METHOD Start : BOOL
VAR_INPUT
END_VAR
bDone := FALSE;
step := 1;
END_METHOD

END_PROGRAM

// ---- POUs/功能塊/Stober驅動/ReadStoberError.TcPOU
PROGRAM ReadStoberError
VAR
	step: INT;
	
	raw_Data	: DWORD;
	
	fb_CoERead : FB_EcCoESdoRead;
	
	readindex : INT;
	
	i_Event :ARRAY [0..17] OF UDINT;
	i_CASE :ARRAY [0..17] OF UDINT;
	
	
	EtherCatAddr	: ARRAY [0..8] OF T_AmsNetId := [9('0.0.0.0.3.1')];
	DriverAddr		: ARRAY [0..8] OF UINT := [1010,1011,1012,1013,1014,1015,1017,1018,1019];
	MoterName		: ARRAY [0..17] OF WSTRING := ["Fx1", "Fx2", "Ax", "Ay", "Az1", "Az2", "Bx", "Bz", "By1", "By2", "Cz1", "Cz2", "Cx", "Cy", "Dy", "Dx", "Dz", "NA"];
	i: INT;
	
	showNumber 		: INT;
END_VAR

CASE step OF
	1:
		fb_CoERead.bExecute		:= FALSE;
		readindex := 0;
		step := step + 1;
		
	2:
		step := 10;
		
	10:
		fb_CoERead.sNetId		:= EtherCatAddr[readindex];
		fb_CoERead.nSlaveAddr	:= DriverAddr[readindex];
		fb_CoERead.nIndex		:= 16#2852;
		fb_CoERead.pDstBuf		:= ADR(raw_Data);
		fb_CoERead.cbBufLen		:= 4;
		fb_CoERead.bExecute		:= TRUE;
		step := step + 1;
		
	11:
		IF NOT fb_CoERead.bBusy THEN
			fb_CoERead.bExecute		:= FALSE;
			step := step + 1;
		END_IF
		
	12:
		IF NOT fb_CoERead.bError THEN
			i_Event[readindex * 2] := DWORD_TO_UDINT(raw_Data);
			step := step + 1;
		ELSE
			step := 0;
		END_IF
	
	13:
		raw_Data := 0;
		step := 20;
		
	20:
		fb_CoERead.nIndex		:= 16#282B;
		fb_CoERead.pDstBuf		:= ADR(raw_Data);
		fb_CoERead.cbBufLen		:= 4;
		fb_CoERead.bExecute		:= TRUE;
		step := step + 1;
		
	21:
		IF NOT fb_CoERead.bBusy THEN
			fb_CoERead.bExecute		:= FALSE;
			step := step + 1;
		END_IF
		
	22:
		IF NOT fb_CoERead.bError THEN
			i_CASE[readindex * 2] := DWORD_TO_UDINT(raw_Data);
			step := step + 1;
		ELSE
			step := 0;
		END_IF
	
	23:
		raw_Data := 0;
		step := 30;
		
	30:
		fb_CoERead.nIndex		:= 16#A852;
		fb_CoERead.pDstBuf		:= ADR(raw_Data);
		fb_CoERead.cbBufLen		:= 4;
		fb_CoERead.bExecute		:= TRUE;
		step := step + 1;
		
	31:
		IF NOT fb_CoERead.bBusy THEN
			fb_CoERead.bExecute		:= FALSE;
			step := step + 1;
		END_IF
		
	32:
		IF NOT fb_CoERead.bError THEN
			i_Event[readindex * 2 + 1] := DWORD_TO_UDINT(raw_Data);
			step := step + 1;
		ELSE
			step := 0;
		END_IF
	
	33:
		raw_Data := 0;
		step := 40;
		
	40:
		fb_CoERead.nIndex		:= 16#A82B;
		fb_CoERead.pDstBuf		:= ADR(raw_Data);
		fb_CoERead.cbBufLen		:= 4;
		fb_CoERead.bExecute		:= TRUE;
		step := step + 1;
		
	41:
		IF NOT fb_CoERead.bBusy THEN
			fb_CoERead.bExecute		:= FALSE;
			step := step + 1;
		END_IF
		
	42:
		IF NOT fb_CoERead.bError THEN
			i_CASE[readindex * 2 + 1] := DWORD_TO_UDINT(raw_Data);
			step := step + 1;
		ELSE
			step := 0;
		END_IF
	
	43:
		raw_Data := 0;
		step := 50;
		
	50:
		IF readindex < 5 THEN
		 	readindex := readindex + 1;
			step := 10;
		ELSE
			readindex := 0;
			step := step + 1;
		END_IF
		
	51:
		step := 60;
		
	60:
		IF showNumber > 0 AND showNumber <= 17 THEN
			i := showNumber - 1;
			step := 61;
		ELSE
			i := 0;
			step := 62;
		END_IF
		
	61:
		pMsg.Push_Info(ErrorCodeConver.StoberErrorCode(MoterName[i], i_Event[i], i_case[i]));
		pMsg.Push_Info(
			WCONCAT(
				STR1:= MoterName[i],
				STR2:= StoberErrorStr(i_Event[i], i_case[i])
		));
		step := 65;
		
	62:
		IF i < 12 AND i <> 8 AND i_Event[i] <> 30 THEN
			pMsg.Push_Info(ErrorCodeConver.StoberErrorCode(MoterName[i], i_Event[i], i_case[i]));
			pMsg.Push_Info(
				WCONCAT(
					STR1:= MoterName[i],
					STR2:= StoberErrorStr(i_Event[i], i_case[i])
			));
		END_IF
		step := step + 1;
		
	63:
		i := i + 1;
		IF i < 12 THEN
			step := step - 1;
		ELSE
			step := 65;
		END_IF
		
	65:
		i := 0;
		step := 90;
		
	90:
		step := 0;
END_CASE

fb_CoERead();

METHOD Read : BOOL
VAR_INPUT
	// 選擇軸
	Axis : AXIS_REF;
END_VAR

step := 1;
END_METHOD

END_PROGRAM

// ---- POUs/功能塊/Stober驅動/StoberErrorStr.TcPOU
FUNCTION StoberErrorStr : WSTRING
VAR_INPUT
	in_Event	: UDINT;
	in_Case		: UDINT;
END_VAR
VAR
END_VAR

CASE in_Event OF
	31:	
		StoberErrorStr := "Short/ground";
		
	32:	
		StoberErrorStr := "Short/ground internal";
		
	33:	
		CASE in_Case OF
			1:
				StoberErrorStr := "Overcurrent(Normal)";
			2:
				StoberErrorStr := "Overcurrent(Fast)";
		END_CASE
		
	34:
		CASE in_Case OF
			1,23,24,25:
				StoberErrorStr := "Hardware fault(FPGA)";
			2:
				StoberErrorStr := "Hardware fault(NOV control unit)";
			3:
				StoberErrorStr := "Hardware fault(NOV-Power Unit)";
			4,5:
				StoberErrorStr := "Hardware fault(Inactive)";
			6:
				StoberErrorStr := "Hardware fault(NOV safety module)";
			7:
				StoberErrorStr := "Hardware fault(Current measurement)";
			8,9,10,11,30:
				StoberErrorStr := "Hardware fault(power supply)";
			12:
				StoberErrorStr := "Hardware fault(Timer control board)";
			13:
				StoberErrorStr := "Hardware fault(Communication module adress-/databus)";
			14:
				StoberErrorStr := "Hardware fault(Communication module signal lines)";
			15:
				StoberErrorStr := "Hardware fault(Communication module clock error)";
			16:
				StoberErrorStr := "Hardware fault(Communication module voltage missing)";
			17:
				StoberErrorStr := "Hardware fault(Communication module databus)";
			18:
				StoberErrorStr := "Hardware fault(Terminal module adress-/databus)";
			19:
				StoberErrorStr := "Hardware fault(Terminal module signal lines)";
			20:
				StoberErrorStr := "Hardware fault(Terminal module clock error)";
			21:
				StoberErrorStr := "Hardware fault(Terminal module voltage is missing)";
			22:
				StoberErrorStr := "Hardware fault(Terminal module databus)";
			26,27,28:
				StoberErrorStr := "Hardware fault(CPU)";
			29:
				StoberErrorStr := "Hardware fault(Communication)";
			31:
				StoberErrorStr := "Hardware fault(Operating unit)";
		END_CASE
		
	35:	
		CASE in_Case OF
			1:
				StoberErrorStr := "Watchdog(Core 0)";
			2:
				StoberErrorStr := "Watchdog(Core 1)";
		END_CASE
		
	36:	
		StoberErrorStr := "High voltage";
		
	37:	
		CASE in_Case OF
			1:
				StoberErrorStr := "Motor encoder(Parameter <-> encoder)";
			2:
				StoberErrorStr := "Motor encoder(Maximum speed)";
			3,5:
				StoberErrorStr := "Motor encoder(AX6)";
			4:
				StoberErrorStr := "Motor encoder(Required AX6)";
			6:
				StoberErrorStr := "Motor encoder(X4 EnDat encoder found)";
			7:
				StoberErrorStr := "Motor encoder(X4 A track/Incremental)";
			8:
				StoberErrorStr := "Motor encoder(X4 no encoder found)";
			10:
				StoberErrorStr := "Motor encoder(X4 A track/Clk)";
			11:
				StoberErrorStr := "Motor encoder(X4 B track/Dat)";
			12:
				StoberErrorStr := "Motor encoder(X4 N track)";
			13:
				StoberErrorStr := "Motor encoder(X4-EnDat alarm)";
			14:
				StoberErrorStr := "Motor encoder(X4 EnDat CRC)";
			15:
				StoberErrorStr := "Motor encoder(X4 double transmission)";
			16:
				StoberErrorStr := "Motor encoder(X4 busy)";
			17:
				StoberErrorStr := "Motor encoder(EBI encoder low battery)";
			18:
				StoberErrorStr := "Motor encoder(EBI encoder battery empty)";
			19:
				StoberErrorStr := "Motor encoder(Alarm bit)";
			20:
				StoberErrorStr := "Motor encoder(Resolver carrier)";
			21:
				StoberErrorStr := "Motor encoder(Low voltage)";
			22:
				StoberErrorStr := "Motor encoder(Resolver sin/cos overvoltage)";
			23,24:
				StoberErrorStr := "Motor encoder(Resolver failure)";
			30:
				StoberErrorStr := "Motor encoder(X120 wire break)";
			35:
				StoberErrorStr := "Motor encoder(X120 double transmission)";
			36:
				StoberErrorStr := "Motor encoder(X120 busy)";
			38:
				StoberErrorStr := "Motor encoder(X120 timeout)";
			43:
				StoberErrorStr := "Motor encoder(X140 EnDat alarm)";
			44:
				StoberErrorStr := "Motor encoder(X140 EnDat CRC)";
			48:
				StoberErrorStr := "Motor encoder(X4 zero pulse missing)";
			49:
				StoberErrorStr := "Motor encoder(X4 zero pulse distance too small)";
			60:
				StoberErrorStr := "Motor encoder(Hiperface synchronisation)";
			61:
				StoberErrorStr := "Motor encoder(Hiperface timeout)";
			62:
				StoberErrorStr := "Motor encoder(Hiperface signal quality)";
			63:
				StoberErrorStr := "Motor encoder(Hiperface link)";
			64:
				StoberErrorStr := "Motor encoder(EnDat3 Timeout)";
			65:
				StoberErrorStr := "Motor encoder(EnDat3 invalid Request)";
			66:
				StoberErrorStr := "Motor encoder(EnDat3 Position Check)";
		END_CASE
		
	38:	
		StoberErrorStr := "Temperature drive controller sensor";
	39:	
		StoberErrorStr := "Temperature drive controller sensor";
		
	40:
		CASE in_Case OF
			1:
				StoberErrorStr := "Invalid data(Fault)";
			2,7:
				StoberErrorStr := "Invalid data(Block missing)";
			3:
				StoberErrorStr := "Invalid data(Data security)";
			4:
				StoberErrorStr := "Invalid data(Checksum)";
			5:
				StoberErrorStr := "Invalid data(Read only)";
			6:
				StoberErrorStr := "Invalid data(Read error)";
			8:
				StoberErrorStr := "Invalid data(Wrong/illegal serial number)";
			9:
				StoberErrorStr := "Invalid data(A00 interrupted - data loss)";
			32:
				StoberErrorStr := "Invalid data(Electronic nameplate)";
			33:
				StoberErrorStr := "Invalid data(Electronic nameplate limit)";
			48:
				StoberErrorStr := "Invalid data(Reverse documentation)";
		END_CASE
		
	41:
		StoberErrorStr := "Temp.MotorTMP";
	24:
		StoberErrorStr := "TempBrakeRes";
	43:
		StoberErrorStr := "AI1 wire break";
	44:
		StoberErrorStr := "External fault 1";
	45:
		StoberErrorStr := "Overtemp.motor i2t";
	46:
		CASE in_Case OF
			1:
				StoberErrorStr := "Low voltage(DC link voltage below limit)";
			2:
				StoberErrorStr := "Low voltage(Failure of one/ all phases (mains))";
			3:
				StoberErrorStr := "Low voltage(Drop in network voltage when power section active)";
		END_CASE
	
	47:
		StoberErrorStr := "Torque/force-max. limit";
	48:
		StoberErrorStr := "Brake release monitoring";
	49:
		CASE in_Case OF
			1:
				StoberErrorStr := "Brake(Brake supply voltage too low)";
			2:
				StoberErrorStr := "Brake(Brake 1: no feedback)";
			3:
				StoberErrorStr := "Brake(Brake 1: short circuit)";
			4:
				StoberErrorStr := "Brake(Brake 1: open load)";
			5:
				StoberErrorStr := "Brake(Brake 2: no feedback)";
			6:
				StoberErrorStr := "Brake(Brake 2: short circuit)";
			7:
				StoberErrorStr := "Brake(Brake 2: open load)";
			8:
				StoberErrorStr := "Brake(F92 switchover not permitted for opened brake)";
			9:
				StoberErrorStr := "Brake(Brake 1 slips)";
			10:
				StoberErrorStr := "Brake(Brake monitoring with engaged brake)";
			11:
				StoberErrorStr := "Brake(Brake monitoring with released brake)";
			12:
				StoberErrorStr := "Brake(Brake monitoring during engaging time)";
			13:
				StoberErrorStr := "Brake(Brake monitoring during release time)";
		END_CASE
	50:
		CASE in_Case OF
			1:
				StoberErrorStr := "Safety module(Inconsistent request (single channel))";
			2:
				StoberErrorStr := "Safety module(Wrong safety module)";
			3:
				StoberErrorStr := "Safety module(Internal error)";
			4:
				StoberErrorStr := "Safety module(PowerUp sequence error)";
			5:
				StoberErrorStr := "Safety module(Wrong interface version)";
			6:
				StoberErrorStr := "Safety module(Fatal error)";
			7:
				StoberErrorStr := "Safety module(Different CRCs in safety config of SafetyModule and DS6)";
			8:
				StoberErrorStr := "Safety module(Safety module startup error)";
			9:
				StoberErrorStr := "Safety module(Safety module failure)";
			10:
				StoberErrorStr := "Safety module(Safety config. missing in ParaModul)";
			11:
				StoberErrorStr := "Safety module(Safety config. from ParaModul activated)";
			12:
				StoberErrorStr := "Safety module(Safety config. missing in Paramodul&safety module)";
			13:
				StoberErrorStr := "Safety module(Safety module activation error)";
			14:
				StoberErrorStr := "Safety module(Command drive to safety module timeout)";
			15:
				StoberErrorStr := "Safety module(Safety module error)";
			16:
				StoberErrorStr := "Safety module(Remove enable!)";
			17:
				StoberErrorStr := "Safety module(Error class LIMIT)";
			18:
				StoberErrorStr := "Safety module(Error class OTHER)";
			19:
				StoberErrorStr := "Safety module(Safety module invalid FSoE address)";
			20:
				StoberErrorStr := "Safety module(Safety control word Error)";
		END_CASE
	51:
		CASE in_Case OF
			1:
				StoberErrorStr := "Virtual master software limit switch(SW-limit switch positive)";
			2:
				StoberErrorStr := "Virtual master software limit switch(SW-limit switch negative)";
			3:
				StoberErrorStr := "Virtual master software limit switch(+/- 31 bit computing limit reached)";
		END_CASE
	52:
		CASE in_Case OF
			1:
				StoberErrorStr := "Communication(CAN Life Guarding Event)";
			2:
				StoberErrorStr := "Communication(CAN Sync Error)";
			3:
				StoberErrorStr := "Communication(CAN Bus Off)";
			4:
				StoberErrorStr := "Communication(PZD-Timeout)";
			5:
				StoberErrorStr := "Communication(Wrong or missing X3 firmware)";
			6:
				StoberErrorStr := "Communication(EtherCAT PDO-Timeout)";
			7:
				StoberErrorStr := "Communication(Reserved)";
			8:
				StoberErrorStr := "Communication(IGB µC failure)";
			9:
				StoberErrorStr := "Communication(IGB serie lost frames)";
			10:
				StoberErrorStr := "Communication(IGB partner serie lost frames)";
			11:
				StoberErrorStr := "Communication(IGB synchronization error)";
			12:
				StoberErrorStr := "Communication(IGB configuration timing)";
			13:
				StoberErrorStr := "Communication(IGB partner synchronization)";
			14:
				StoberErrorStr := "Communication(PZD parameter figure faulty)";
			15:
				StoberErrorStr := "Communication(Wrong firmware for applicataion)";
			16:
				StoberErrorStr := "Communication(PROFINET Sign-of-Life synchronisation failed)";
		END_CASE
	53:
		CASE in_Case OF
			1:
				StoberErrorStr := "Limit switch(Hardware-Limit-Switch positive)";
			2:
				StoberErrorStr := "Limit switch(Hardware-Limit-Switch negative)";
			3:
				StoberErrorStr := "Limit switch(SW-limit switch positive)";
			4:
				StoberErrorStr := "Limit switch(SW-limit switch negative)";
			5:
				StoberErrorStr := "Limit switch(+/- 31 bit computing limit reached)";
			6:
				StoberErrorStr := "Limit switch(Linear motor moving range)";
			7:
				StoberErrorStr := "Limit switch(Both limit switches not connected)";
		END_CASE
	54:
		StoberErrorStr := "Following error";
	55:
		CASE in_Case OF
			1:
				StoberErrorStr := "Option module(Communication module wrong/missing)";
			2:
				StoberErrorStr := "Option module(EC6 failure)";
			3:
				StoberErrorStr := "Option module(CA6 failure)";
			4:
				StoberErrorStr := "Option module(DP6 failure)";
			5:
				StoberErrorStr := "Option module(PN6 failure)";
			6:
				StoberErrorStr := "Option module(Communication module incompatible)";
			7:
				StoberErrorStr := "Option module(Terminal module wrong/ missing)";
			8:
				StoberErrorStr := "Option module(IO6 failure)";
			9:
				StoberErrorStr := "Option module(RI6 failure)";
			10:
				StoberErrorStr := "Option module(XB6 failure)";
			11:
				StoberErrorStr := "Option module(XB6 encoder simulation initialization)";
			12:
				StoberErrorStr := "Option module(XB6 24V supply)";
			13:
				StoberErrorStr := "Option module(Terminal module incompatible)";
		END_CASE
	56:
		CASE in_Case OF
			1:
				StoberErrorStr := "Overspeed(Motor encoder)";
			2:
				StoberErrorStr := "Overspeed(Position encoder)";
			3:
				StoberErrorStr := "Overspeed(Motor & position encoder)";
		END_CASE
	57:
		CASE in_Case OF
			1:
				StoberErrorStr := "Runtime requirement(RT0)";
			2:
				StoberErrorStr := "Runtime requirement(RT2)";
			3:
				StoberErrorStr := "Runtime requirement(RT3)";
			4:
				StoberErrorStr := "Runtime requirement(RT4)";
			5:
				StoberErrorStr := "Runtime requirement(RT5)";
			6:
				StoberErrorStr := "Runtime requirement(RT2 (Core1))";
			7:
				StoberErrorStr := "Runtime requirement(RT4 (Core1))";
		END_CASE
	58:
		CASE in_Case OF
			1:
				StoberErrorStr := "Encoder simulation(Maximum speed)";
			2:
				StoberErrorStr := "Encoder simulation(Timeout)";
			3:
				StoberErrorStr := "Encoder simulation(X120 wire break)";
		END_CASE
	
	59:
		StoberErrorStr := "Overtemperature drive controller i2t";
	60:
		StoberErrorStr := "Application event 0";
	61:
		StoberErrorStr := "Application event 1";
	62:
		StoberErrorStr := "Application event 2";
	63:
		StoberErrorStr := "Application event 3";
	64:
		StoberErrorStr := "Application event 4";
	65:
		StoberErrorStr := "Application event 5";
	66:
		StoberErrorStr := "Application event 6";
	67:
		StoberErrorStr := "Application event 7";
	68:
		StoberErrorStr := "External fault 2";
	69:
		CASE in_Case OF
			1:
				StoberErrorStr := "Motor connection(Motor not disconnected)";
			2:
				StoberErrorStr := "Motor connection(No motor connected)";
			3:
				StoberErrorStr := "Motor connection(Wake and Shake failed)";
			4:
				StoberErrorStr := "Motor connection(Brake)";
		END_CASE
	70:
		CASE in_Case OF
			1:
				StoberErrorStr := "Parameter consistency(Wrong encoder model)";
			2:
				StoberErrorStr := "Parameter consistency(X120 data direction)";
			3:
				StoberErrorStr := "Parameter consistency(B12<->B20)";
			4:
				StoberErrorStr := "Parameter consistency(B10<->H31)";
			5:
				StoberErrorStr := "Parameter consistency(Negative slip frequency)";
			6:
				StoberErrorStr := "Parameter consistency(Torque limit too high)";
			7:
				StoberErrorStr := "Parameter consistency(SSI passive)";
			8:
				StoberErrorStr := "Parameter consistency(v-max (I10) exeeds maximum (B83))";
			9:
				StoberErrorStr := "Parameter consistency(E102/E103 missing)";
			10:
				StoberErrorStr := "Parameter consistency(G104 <-> G27)";
			11:
				StoberErrorStr := "Parameter consistency(Reference retaining)";
			12:
				StoberErrorStr := "Parameter consistency(Type of axis)";
			13:
				StoberErrorStr := "Parameter consistency(Motor temperature sensor)";
			14:
				StoberErrorStr := "Parameter consistency(Max. acceleration I11>B143)";
			15:
				StoberErrorStr := "Parameter consistency(Safety watchdog time)";
			16:
				StoberErrorStr := "Parameter consistency(I10 > C11)";
		END_CASE
	71:
		CASE in_Case OF
			1:
				StoberErrorStr := "Firmware(Firmware defective)";
			2:
				StoberErrorStr := "Firmware(Activate firmware!)";
			3:
				StoberErrorStr := "Firmware(CRC-error)";
			4:
				StoberErrorStr := "Firmware(CPU)";
		END_CASE
	72:
		CASE in_Case OF
			1:
				StoberErrorStr := "Brake test timeout(B311timeout:B300 mandatory)";
			2:
				StoberErrorStr := "Brake test timeout(Brake defective:B300 mandatory)";
			3:
				StoberErrorStr := "Brake test timeout(Brake test necessary)";
		END_CASE
	73:
		CASE in_Case OF
			1:
				StoberErrorStr := "Axis 2 brake test timeout(B311timeout:B300 mandatory)";
			2:
				StoberErrorStr := "Axis 2 brake test timeout(Brake defective:B300 mandatory)";
			3:
				StoberErrorStr := "Axis 2 brake test timeout(Brake test necessary)";
		END_CASE
	74:
		CASE in_Case OF
			1:
				StoberErrorStr := "Axis 3 brake test timeout(B311timeout:B300 mandatory)";
			2:
				StoberErrorStr := "Axis 3 brake test timeout(Brake defective:B300 mandatory)";
			3:
				StoberErrorStr := "Axis 3 brake test timeout(Brake test necessary)";
			
		END_CASE
	75:
		CASE in_Case OF
			1:
				StoberErrorStr := "Axis 4 brake test timeout(B311timeout:B300 mandatory)";
			2:
				StoberErrorStr := "Axis 4 brake test timeout(Brake defective:B300 mandatory)";
			3:
				StoberErrorStr := "Axis 4 brake test timeout(Brake test necessary)";
		END_CASE
	76:
		CASE in_Case OF
			1:
				StoberErrorStr := "Position encoder(Parameter <-> encoder)";
			2:
				StoberErrorStr := "Position encoder(Maximum speed)";
			3:
				StoberErrorStr := "Position encoder(AX6)";
			4:
				StoberErrorStr := "Position encoder(Required AX6)";
			5:
				StoberErrorStr := "Position encoder(AX6)";
			6:
				StoberErrorStr := "Position encoder(X4 EnDat encoder found)";
			7:
				StoberErrorStr := "Position encoder(X4 A track/Incremental)";
			8:
				StoberErrorStr := "Position encoder(X4 no encoder found)";
			9:
				StoberErrorStr := "Position encoder(Referencing failed)";
			10:
				StoberErrorStr := "Position encoder(X4 A track/Clk)";
			11:
				StoberErrorStr := "Position encoder(X4 B track/Dat)";
			12:
				StoberErrorStr := "Position encoder(X4 N track)";
			13:
				StoberErrorStr := "Position encoder(X4-EnDat alarm)";
			14:
				StoberErrorStr := "Position encoder(X4 EnDat CRC)";
			15:
				StoberErrorStr := "Position encoder(X4 double transmission)";
			16:
				StoberErrorStr := "Position encoder(X4 busy)";
			17:
				StoberErrorStr := "Position encoder(EBI encoder low battery)";
			18:
				StoberErrorStr := "Position encoder(EBI encoder battery empty)";
			19:
				StoberErrorStr := "Position encoder(Alarm bit)";
			20:
				StoberErrorStr := "Position encoder(Resolver carrier)";
			21:
				StoberErrorStr := "Position encoder(Resolver sin/cos undervoltage)";
			22:
				StoberErrorStr := "Position encoder(Resolver sin/cos overvoltage)";
			23,24:
				StoberErrorStr := "Position encoder(Resolver failure)";
			30:
				StoberErrorStr := "Position encoder(X120 wire break)";
			35:
				StoberErrorStr := "Position encoder(X120 double transmission)";
			36:
				StoberErrorStr := "Position encoder(X120 busy)";
			38:
				StoberErrorStr := "Position encoder(X120 timeout)";
			43:
				StoberErrorStr := "Position encoder(X140 EnDat alarm)";
			44:
				StoberErrorStr := "Position encoder(X140 EnDat CRC)";
			48:
				StoberErrorStr := "Position encoder(X4 zero pulse missing)";
			49:
				StoberErrorStr := "Position encoder(X4 zero pulse distance too small)";
			60:
				StoberErrorStr := "Position encoder(Hiperface synchronisation)";
			61:
				StoberErrorStr := "Position encoder(Hiperface timeout)";
			62:
				StoberErrorStr := "Position encoder(Hiperface signal quality)";
			63:
				StoberErrorStr := "Position encoder(Hiperface link)";
			64:
				StoberErrorStr := "Position encoder(EnDat3 Timeout)";
			65:
				StoberErrorStr := "Position encoder(EnDat3 invalid Request)";
			66:
				StoberErrorStr := "Position encoder(EnDat3 Position Check)";
		END_CASE
	77:
		CASE in_Case OF
			1:
				StoberErrorStr := "Master encoder(Parameter <-> encoder)";
			2:
				StoberErrorStr := "Master encoder(Maximum speed)";
			3:
				StoberErrorStr := "Master encoder(AX6)";
			4:
				StoberErrorStr := "Master encoder(Required AX6)";
			5:
				StoberErrorStr := "Master encoder(AX6)";
			6:
				StoberErrorStr := "Master encoder(X4 EnDat encoder found)";
			7:
				StoberErrorStr := "Master encoder(X4 A track/Incremental)";
			8:
				StoberErrorStr := "Master encoder(X4 no encoder found)";
			10:
				StoberErrorStr := "Master encoder(X4 A track/Clk)";
			11:
				StoberErrorStr := "Master encoder(X4 B track/Dat)";
			12:
				StoberErrorStr := "Master encoder(X4 N track)";
			13:
				StoberErrorStr := "Master encoder(X4-EnDat alarm)";
			14:
				StoberErrorStr := "Master encoder(X4 EnDat CRC)";
			15:
				StoberErrorStr := "Master encoder(X4 double transmission)";
			16:
				StoberErrorStr := "Master encoder(X4 busy)";
			19:
				StoberErrorStr := "Master encoder(Alarm bit)";
			20:
				StoberErrorStr := "Master encoder(Resolver carrier)";
			21:
				StoberErrorStr := "Master encoder(Resolver sin/cos undervoltage)";
			22:
				StoberErrorStr := "Master encoder(Resolver sin/cos overvoltage)";
			23:
				StoberErrorStr := "Master encoder(Resolver failure)";
			24:
				StoberErrorStr := "Master encoder(Resolver failure)";
			30:
				StoberErrorStr := "Master encoder(X120 wire break)";
			35:
				StoberErrorStr := "Master encoder(X120 double transmission)";
			36:
				StoberErrorStr := "Master encoder(X120 busy)";
			38:
				StoberErrorStr := "Master encoder(X120 timeout)";
			43:
				StoberErrorStr := "Master encoder(X140 EnDat alarm)";
			44:
				StoberErrorStr := "Master encoder(X140 EnDat CRC)";
			50:
				StoberErrorStr := "Master encoder(Source of position missing)";
			51:
				StoberErrorStr := "Master encoder(Timestamp source missing)";
		END_CASE
	78:
		CASE in_Case OF
			1:
				StoberErrorStr := "Position limit cyclic(Illegal direction)";
			2:
				StoberErrorStr := "Position limit cyclic(Reference value invalid)";
			3:
				StoberErrorStr := "Position limit cyclic(Extrapolation time I423 exceeded)";
		END_CASE
	79:
		StoberErrorStr := "Motor/position encoder plausibility";
	80:
		CASE in_Case OF
			1:
				StoberErrorStr := "Illegal action(Brake)";
			2:
				StoberErrorStr := "Illegal action(Brake)";
		END_CASE
	81:
		CASE in_Case OF
			1:
				StoberErrorStr := "Motor allocation(Different motor type)";
			32:
				StoberErrorStr := "Motor allocation(Different motor)";
			33:
				StoberErrorStr := "Motor allocation(Different motor & brake)";
			34:
				StoberErrorStr := "Motor allocation(Different motor & temperature sensor)";
			35:
				StoberErrorStr := "Motor allocation(Different motor & brake & temperature sensor)";
			36:
				StoberErrorStr := "Motor allocation(Different motor & gear unit)";
			37:
				StoberErrorStr := "Motor allocation(Different motor, brake & gear unit)";
			38:
				StoberErrorStr := "Motor allocation(Different motor, temperature sensor & gear unit)";
			39:
				StoberErrorStr := "Motor allocation(Different motor, brake, temperature sensor & gear unit)";
			64:
				StoberErrorStr := "Motor allocation(Different commutation)";
			65:
				StoberErrorStr := "Motor allocation(Different commutation & brake)";
			66:
				StoberErrorStr := "Motor allocation(Different commutation & temperature sensor)";
			67:
				StoberErrorStr := "Motor allocation(Different commutation & brake & temperature sensor)";
			129:
				StoberErrorStr := "Motor allocation(Different brake)";
			130:
				StoberErrorStr := "Motor allocation(Different temperature sensor)";
			131:
				StoberErrorStr := "Motor allocation(Different brake & temperature sensor)";
			150:
				StoberErrorStr := "Motor allocation(Temperature sensor unknown)";
			
		END_CASE
	82:
		CASE in_Case OF
			1:
				StoberErrorStr := "Hall sensor(Invalid sample)";
			2:
				StoberErrorStr := "Hall sensor(Invalid sequence)";
			3:
				StoberErrorStr := "Hall sensor(Signal edge missing)";
			4:
				StoberErrorStr := "Hall sensor(X120 wire break)";
		END_CASE
	83:
		StoberErrorStr := "Failure of one/ all phases (mains)";
	84:
		StoberErrorStr := "Drop in network voltage when power section active";
	85:
		CASE in_Case OF
			1:
				StoberErrorStr := "Excessive jump in reference value(Position)";
			2:
				StoberErrorStr := "Excessive jump in reference value(Velocity)";
		END_CASE
	86:
		CASE in_Case OF
			1:
				StoberErrorStr := "Unknown LeanMotor(Motor)";
			2:
				StoberErrorStr := "Unknown LeanMotor(Cable length)";
		END_CASE
	87:
		StoberErrorStr := "Reference lostReference loss";
	88:
		StoberErrorStr := "Control panel";
	89:
		CASE in_Case OF
			1:
				StoberErrorStr := "Maximum current LM(Id)";
			2:
				StoberErrorStr := "Maximum current LM(Iq)";
		END_CASE
	90:
		CASE in_Case OF
			1:
				StoberErrorStr := "Motion block(Next motion block missing)";
			2:
				StoberErrorStr := "Motion block(Target Position in reverse direction)";
		END_CASE
	91:
		StoberErrorStr := "PM geared motor replacement";
	
END_CASE

END_FUNCTION

// ---- POUs/硬體控制/軸/AxisFx.TcPOU
FUNCTION_BLOCK AxisFx EXTENDS MultipleAxisBase IMPLEMENTS I_Axis
VAR_INPUT
END_VAR
VAR_OUTPUT
END_VAR
VAR
	fb_SetPosition : MC_SetPosition;
END_VAR

(* =================== 繼承至 AxisBase ===================*)

// 確定兩個軸都有映射才執行
IF __ISVALIDREF(Axis1) THEN
	b_ISVALIDREF := TRUE;
	Main();
	Step1_13_SetPos();
END_IF

ACTION MC_FB:
// 正轉極限
Axis1Power.Enable_Positive:= OutLimiter;
Axis2Power.Enable_Positive:= OutLimiter;
// 反轉極限
Axis1Power.Enable_Negative:= inLimiter;
Axis2Power.Enable_Negative:= inLimiter;

Axis1.ReadStatus();
Axis2.ReadStatus();

// 軸速度百分比

IF hmi.Auto_Pause THEN
	Axis1Power.Override := 0;
ELSE
	Axis1Power.Override := Axis.Override;
END_IF

Axis2Power.Override := Axis.Override;

(*===================== 軸電源 =====================*)
Axis1Power(Axis:= Axis1);
Axis2Power(Axis:= Axis2);

(*===================== 軸重置 =====================*)
Axis1Reset(Axis:= Axis1);
Axis2Reset(Axis:= Axis2);

(*===================== 軸耦合 =====================*)
AxisGearIn(master := Axis1, slave := Axis2);

(*===================== 軸解耦 =====================*)
AxisGearOut(slave := Axis2);

(*===================== 軸停止 =====================*)
Axis1Stop(Axis:= Axis1);

(*===================== 軸命令取消 =====================*)
Axis1Halt(Axis:= Axis1);

(*===================== 軸絕對移動 =====================*)
fb_AbsMove(Axis:= Axis1);

(*===================== 軸相對移動 =====================*)
fb_RelMove(Axis:= Axis1);

(*===================== 軸歸零 =====================*)
fb_Axis1_NcIoOutput(Axis:= Axis1, Device := NcIoDeviceDrive, NcIoOutput := NcIoOutputnCtrl2);
fb_Axis2_NcIoOutput(Axis:= Axis2, Device := NcIoDeviceDrive, NcIoOutput := NcIoOutputnCtrl2);

(*===================== 軸歸零 =====================*)
fb_Home(Axis:= Axis1, HomingMode:= MC_Direct);

(*===================== 軸設定位置 =====================*)
fb_SetPosition.Options.ClearPositionLag := TRUE;
fb_SetPosition(Axis:= Axis1, Mode := FALSE);

(*===================== 軸寫入BOOL參數 =====================*)
fb_WriteBoolParameter(Axis:= Axis1);

(*===================== 軸寫入參數 =====================*)
fb_WriteParameter(Axis:= Axis1);

(*===================== 背隙補償 =====================*)
fb_BacklashCompensation(Axis:= Axis1);
END_ACTION

METHOD SetPos : BOOL
VAR_INPUT
	Pos : LREAL;
END_VAR
TargetPos := pos;

// ============ 紀錄啟動條件 ============
_log.fbJson.StartObject();
_log.fbJson.AddKeyString('MethodName','SetPos');
_log.fbJson.AddKeyLreal('Position', Pos);
_log.JsonOutput();
// ======================================

step:=1300;
END_METHOD

ACTION Step1_13_SetPos:
(*========================================
				歸零
=========================================*)	
CASE step OF
	1300:
		fb_SetPosition.Execute := FALSE;
		step := step + 1;
		
	1301: 
		step:= 1350;
			
		
	1350:// 設定原點
		fb_SetPosition.Position := TargetPos;
		fb_SetPosition.Execute := TRUE;
		step:=step + 1;
		
	1351:
		IF fb_SetPosition.Busy OR fb_SetPosition.Error THEN
			step:=step + 1;
		END_IF
		
	1352:
		IF fb_SetPosition.Done THEN
			fb_SetPosition.Execute := FALSE;
			step:=step + 1;
		ELSIF fb_SetPosition.Error THEN
			pMsg.Push_Error(
				ErrorCodeConver.Str(str0:= scAxisName, str1:= ":位置同步失敗", str2:= ws_step, ErrorCode:= fb_SetPosition.ErrorID)
			);
			fb_SetPosition.Execute := FALSE;
			step:=step + 10000;
		END_IF
		
	
	1353:
		step:= 1390;
	
			
	1390:
		bDone := TRUE;
		step:=890;
END_CASE
END_ACTION

ACTION Step1_3_Home:
(*========================================
				歸零
=========================================*)	
CASE step OF
	300:
		fb_Home.Execute := FALSE;
		step := step + 1;
		
	301: 
		Origin_pos := Pos;
		step:= 350;
			
		
	350:// 設定原點
		fb_Home.Execute := TRUE;
		step:=step + 1;
		
	351:
		IF fb_Home.Busy OR fb_Home.Error THEN
			step:=step + 1;
		END_IF
		
	352:
		IF fb_Home.Done THEN
			fb_Home.Execute := FALSE;
			bHome := TRUE;
			step:=step + 1;
		ELSIF fb_Home.Error THEN
			pMsg.Push_Error(
				ErrorCodeConver.Str(str0:= scAxisName, str1:= ":位置清除失敗", str2:= ws_step, ErrorCode:= fb_Home.ErrorID)
			);
			fb_Home.Execute := FALSE;
			step:=step + 10000;
		END_IF
		
	
	353:
		tmr200.in :=TRUE;
		IF tmr200.q THEN
			tmr200.in :=FALSE;
			step:=step + 1;
		END_IF
		
	354:
		step:= 360;
		
	360:
		step:= 390;
	
			
	390://延遲
		tmr200.in :=TRUE;
		IF tmr200.q THEN
			tmr200.in :=FALSE;
			bDone := TRUE;
			step:=890;
		END_IF
END_CASE
END_ACTION

END_FUNCTION_BLOCK

// ---- POUs/硬體控制/軸/MultipleAxisBase.TcPOU
FUNCTION_BLOCK MultipleAxisBase EXTENDS AxisBase IMPLEMENTS I_Axis
VAR_INPUT
	Axis2 : REFERENCE TO AXIS_REF;
END_VAR
VAR_OUTPUT
END_VAR
VAR
	
(*==============================================
				MC 功能快
==============================================*)
	Axis2Power	: MC_Power;
	Axis2Reset	: MC_Reset;
	
	AxisGearIn	: MC_GearIn;
	AxisGearOut : MC_GearOut;
	
	fb_Axis2_NcIoOutput : MC_WriteNcIoOutput;
(*==============================================*)
	scAxisName2 : wstring;
	
END_VAR

(* =================== 繼承至 AxisBase ===================*)

// 確定兩個軸都有映射才執行
IF __ISVALIDREF(Axis1) AND __ISVALIDREF(Axis2) THEN
	b_ISVALIDREF := TRUE;
	Main();
END_IF

ACTION MC_FB:
// 正轉極限
Axis1Power.Enable_Positive:= OutLimiter;
Axis2Power.Enable_Positive:= OutLimiter;
// 反轉極限
Axis1Power.Enable_Negative:= inLimiter;
Axis2Power.Enable_Negative:= inLimiter;

Axis1.ReadStatus();
Axis2.ReadStatus();

// 軸速度百分比

IF hmi.Auto_Pause THEN
	Axis1Power.Override := 0;
ELSE
	Axis1Power.Override := Axis.Override;
END_IF

Axis2Power.Override := Axis.Override;

(*===================== 軸電源 =====================*)
Axis1Power(Axis:= Axis1);
Axis2Power(Axis:= Axis2);

(*===================== 軸重置 =====================*)
Axis1Reset(Axis:= Axis1);
Axis2Reset(Axis:= Axis2);

(*===================== 軸耦合 =====================*)
AxisGearIn(master := Axis1, slave := Axis2);

(*===================== 軸解耦 =====================*)
AxisGearOut(slave := Axis2);

(*===================== 軸停止 =====================*)
Axis1Stop(Axis:= Axis1);

(*===================== 軸命令取消 =====================*)
Axis1Halt(Axis:= Axis1);

(*===================== 軸絕對移動 =====================*)
fb_AbsMove(Axis:= Axis1);

(*===================== 軸相對移動 =====================*)
fb_RelMove(Axis:= Axis1);

(*===================== 軸歸零 =====================*)
fb_Axis1_NcIoOutput(Axis:= Axis1, Device := NcIoDeviceDrive, NcIoOutput := NcIoOutputnCtrl2);
fb_Axis2_NcIoOutput(Axis:= Axis2, Device := NcIoDeviceDrive, NcIoOutput := NcIoOutputnCtrl2);

(*===================== 軸歸零 =====================*)
fb_Home(Axis:= Axis1, HomingMode:= MC_Direct);

(*===================== 軸寫入BOOL參數 =====================*)
fb_WriteBoolParameter(Axis:= Axis1);

(*===================== 軸寫入參數 =====================*)
fb_WriteParameter(Axis:= Axis1);

(*===================== 背隙補償 =====================*)
fb_BacklashCompensation(Axis:= Axis1);
END_ACTION

PROPERTY Name2 : WSTRING
GET
Name2 := scAxisName2;
END_GET
SET
scAxisName2 := Name2;
END_SET
END_PROPERTY

ACTION Step0_Start:
	(*============================
				啟動馬達
	  ============================*)
CASE step OF
	
	1://開始移動流程
		// 設定狀態
		bDone := FALSE;
		tmrWdt.IN := FALSE;
// 		SetDyn(bJogMode);
		Axis1Reset.Execute :=FALSE;
		Axis2Reset.Execute :=FALSE;
		AxisGearIn.Execute := FALSE;
		IF NOT bDone THEN
			step := 10;
		END_IF
		
	10:
		IF axis1.Status.Error OR axis2.Status.Error THEN
			step := step + 1;
		ELSE
			step := 20;
		END_IF
		
	11:
		IF axis1.Status.Error THEN
			Axis1Reset.Execute :=TRUE;
			step := step + 1;
		ELSE
			step := 13;
		END_IF
		
		
	12:
		IF NOT axis1.Status.Error AND Axis1Reset.Done THEN
			Axis1Reset.Execute :=FALSE;
			step := step + 1;
		ELSIF Axis1Reset.Error THEN
			pMsg.Push_Error(
				ErrorCodeConver.Str(str0:= scAxisName, str1:= ": 馬達無法重置", ErrorCode:= Axis1Reset.ErrorID)
			);
			Axis1Reset.Execute :=FALSE;
			step:=step + 10000;
		END_IF
		
	13:
		IF axis2.Status.Error THEN
			Axis2Reset.Execute :=TRUE;
			step := step + 1;
		ELSE
			step := 15;
		END_IF
		
		
	14:
		IF NOT axis2.Status.Error AND Axis2Reset.Done THEN
			Axis2Reset.Execute :=FALSE;
			step := step + 1;
		ELSIF Axis2Reset.Error THEN
			pMsg.Push_Error(
				ErrorCodeConver.Str(str0:= scAxisName, str1:= ":馬達無法重置", ErrorCode:= Axis2Reset.ErrorID)
			);
			Axis2Reset.Execute :=FALSE;
			step:=step + 10000;
		END_IF
		
	15:
		step := 20;

		
	20: // 檢查馬達1是否已啟動
		IF NOT Axis1Power.Status  THEN
			step := step + 1;
		ELSE
			step := 24;
		END_IF
		
	21:// 啟動馬達1
		Axis1Power.Enable := TRUE;
		tmrWdt.IN := TRUE;
		step := step + 1;
		
	22:// 等待馬達啟動完成
		IF Axis1Power.Status THEN
			step := step + 1;
			tmrWdt.IN := FALSE;
			
		ELSIF tmrWdt.Q OR Axis1Power.Error THEN
			tmrWdt.IN := FALSE;
			IF _retry_count > 3 THEN
				pMsg.Push_Error(ErrorCodeConver.Str(
					str0:= scAxisName, str1:= ": 馬達1啟動失敗", ErrorCode:= Axis1Power.ErrorID)
				);
				step:=step + 10000;
			ELSE
				Axis1Power.Enable := FALSE;
				_retry_count := _retry_count + 1;
				step := 10;
			END_IF
		END_IF
		
	23:// 馬達啟動後延遲
		tmr1.in:=TRUE;
		IF tmr1.Q THEN
			tmr1.IN:=FALSE;
			step := step + 1;
		END_IF
		
	24: // 啟動馬達2
		Axis2Power.Enable := TRUE;
		tmrWdt.IN := TRUE;
		step := step + 1;
		
	25:// 等待馬達啟動完成
		IF Axis2Power.Status THEN
			step := step + 1;
			tmrWdt.IN := FALSE;
			
		ELSIF tmrWdt.Q OR Axis2Power.Error THEN
			tmrWdt.IN := FALSE;
			IF _retry_count > 3 THEN
				pMsg.Push_Error(
					ErrorCodeConver.Str(str0:= scAxisName, str1:= ": 馬達2達啟動失敗", ErrorCode:= Axis2Power.ErrorID)
				);
				step:=step + 10000;
			ELSE
				Axis2Power.Enable := FALSE;
				_retry_count := _retry_count + 1;
				step := 10;
			END_IF
		END_IF
		
	26:// 馬達啟動後延遲
		tmr1.in:=TRUE;
		IF tmr1.Q THEN
			tmr1.IN:=FALSE;
			step:=50;
		END_IF
		
	40:
		fb_BacklashCompensation.Enable := FALSE;
		step := step + 1;
		
	41:
		// 背隙值 (mm)
		fb_BacklashCompensation.Backlash := 0.05;
		// 正向補償 (往正方向移動時補償，預設是反方向移動時補償)
		fb_BacklashCompensation.CompensationInPositiveDirection := FALSE;
		// 背隙補償的速度 (mm/s)
		fb_BacklashCompensation.Ramp := 1;
		// 解除時機
		fb_BacklashCompensation.DisableMode  := E_DisableMode.DisableModeReset;
		// 功能啟動
		fb_BacklashCompensation.Enable := TRUE;
		step := step + 1;
		
	42:
		IF fb_BacklashCompensation.Enabled THEN
			step := step + 1;
		ELSIF fb_BacklashCompensation.Error THEN
			fb_BacklashCompensation.Enable := FALSE;
			step := step + 1;
		END_IF
		
	43:
		step := 50;
			
		
	50:
		IF axis2.Status.Coupled THEN
			step := 60;
		ELSE
			step := step + 1;
		END_IF 

	51: // 軸耦合
		AxisGearIn.RatioNumerator := 1;
		AxisGearIn.RatioDenominator := 1;
		AxisGearIn.Execute := TRUE;
		step := step + 1;
		
	52:
		IF AxisGearIn.InGear THEN
			AxisGearIn.Execute := FALSE;
			step := step + 1;
		ELSIF AxisGearIn.Error THEN
			pMsg.Push_Error(
				ErrorCodeConver.Str(str0:= scAxisName, str1:= ": 耦合失敗", ErrorCode:= AxisGearIn.ErrorID)
			);
			AxisGearIn.Execute := FALSE;
			step := step + 10000;
		END_IF
		
	53:
		step := 60;
		
	60: //模式選擇
		CASE Mode OF
			ActionMode.DoNothing:
				bdone := TRUE;
				step := 0;
			
			ActionMode.AbsMove:
				step := 100;
				
			ActionMode.RelMove:
				step := 200;
				
			ActionMode.Home:
				step := 300;
		END_CASE
		
END_CASE
END_ACTION

ACTION Step8_End:
	(*======================================
					關閉馬達
	  ======================================*)
CASE step OF
	// ============== 停止 + 關閉==============
	800:
		Axis1Reset.Execute	:= FALSE;
		Axis1Stop.Execute	:= FALSE;
		Axis1Halt.Execute	:= FALSE;
		fb_AbsMove.Execute	:= FALSE;
		fb_RelMove.Execute	:= FALSE;
		fb_Home.Execute		:= FALSE;
		Axis1Stop.Execute	:= FALSE;
		step := step + 1;
		
	801:
		IF Axis1.Status.Moving THEN
			step := step + 1;
		ELSE
			step := 810;
		END_IF
	
	802:
		Axis1Stop.Execute := TRUE;
		step := step + 1;
		
	803:
		Axis1Stop.Execute := TRUE;
		step := step + 1;
		
	804:
		IF Axis1Stop.Done OR Axis1Stop.Error THEN
			Axis1Stop.Execute := FALSE;
			step := step + 1;
		END_IF
		
	805:
		tmr800.PT := T#1S;
		tmr800.in:=TRUE;
		IF tmr800.Q THEN
			tmr800.IN:=FALSE;
			step := step + 1;
		END_IF
		
	806:
		step:=810;
		
	
	810:
		Axis1Power.Enable := FALSE;
		IF Axis1.Status.Disabled THEN
			step := step + 1;
		END_IF
		
	811:
		Axis2Power.Enable := FALSE;
		IF Axis2.Status.Disabled THEN
			step := step + 1;
		END_IF
			
	812:// 馬達關閉後延遲
		tmr800.in:=TRUE;
		IF tmr800.Q THEN
			tmr800.IN:=FALSE;
			step := step + 1;
		END_IF
		
	813:
		Mode := ActionMode.DoNothing;
		step:=820;
		
	820:
		IF axis2.Status.Coupled THEN
			step := step + 1;
		ELSE
			step := 890;
		END_IF
		
	821:
		AxisGearOut.Execute := TRUE;
		step := step + 1;
		
	822:
		IF AxisGearOut.Done OR AxisGearOut.Error THEN
			AxisGearOut.Execute := FALSE;
			step := step + 1;
		END_IF
		
	823:
		step:=890;
		
		
// ==============停止==============
	850:
		Axis1Stop.Deceleration := Dec;
		Axis1Stop.Jerk := Dec * 5;
		Axis1Stop.Execute := FALSE;
		step := step + 1;
	
	851:
		Axis1Stop.Execute := TRUE;
		step := step + 1;
		
	852:
		IF Axis1Stop.Done OR Axis1Stop.Error THEN
			Axis1Stop.Execute := FALSE;
			step := step + 1;
		END_IF
		
	853:
		tmr800.PT := T#1S;
		tmr800.in:=TRUE;
		IF tmr800.Q THEN
			tmr800.IN:=FALSE;
			step := step + 1;
		END_IF
		
	854:
		step:=890;
		
		
			
	890:// 結束程式
		Mode := ActionMode.DoNothing;
		step:=0;

END_CASE
END_ACTION

END_FUNCTION_BLOCK

// ---- POUs/硬體控制/軸/AxisBase.TcPOU
FUNCTION_BLOCK AxisBase IMPLEMENTS I_Axis
VAR_INPUT
END_VAR
VAR_OUTPUT
END_VAR
VAR
	// 模式
	Mode: ActionMode;
	// 步進
	step: INT;
	stepA: INT;
	// 發生錯誤步
	ws_step: WSTRING;
	// 目標位置
	TargetPos: LREAL;
	// 動作速度
	Velocity: LREAL;
	// 動作減速度
	Dec : LREAL := 0;
(*=======================================
				計時器
=======================================*)
	
	tmr1: TON := (PT := TIME#100MS);
	tmr2: TON := (PT := TIME#100MS);
	tmr100: TON;
	tmr200: TON := (PT := TIME#1S);
	tmr201: TON := (PT := TIME#1S);
	tmr800: TON := (PT := TIME#100MS);
	
	// 超時監視計時器
	tmrWdt: Ton := (PT := TIME#10S0MS);
  	
	
(*=======================================
				軸IO
=======================================*)

	
	Estop_Old: BOOL;
	
	Estop_Trig : R_TRIG;

(*==============================================
					MC 功能快
==============================================*)
	

	Axis1Power	: MC_Power;
	Axis1Reset	: MC_Reset;
	Axis1Stop	: MC_Stop;
	Axis1Halt	: MC_Halt;
	
	fb_AbsMove	: MC_MoveAbsolute;
	fb_RelMove	: MC_MoveRelative;
	fb_Home		: MC_Home;
	fb_BacklashCompensation	: MC_BacklashCompensation;
	
	fb_Axis1_NcIoOutput : MC_WriteNcIoOutput;
	
	
	fb_WriteBoolParameter : MC_WriteBoolParameterPersistent;
	fb_WriteParameter: MC_WriteParameterPersistent;
(*==============================================*)

	Origin_pos: LREAL;
	
	// 軸名稱
	scAxisName : WSTRING;
	
	// 運動距離
	total_Move : POINTER TO LREAL;
	
	
	move_Start_Pos : LREAL;
	move_RTrig : R_TRIG;
	move_FTrig : F_TRIG;
	_retry_count: INT;

	_log : Step_Log;
END_VAR

VAR_OUTPUT
	// 功能執行中
	bBuzy 	: BOOL;
	// 功能結束
	bDone	: BOOL;
	// 發生錯誤
	bError	: BOOL;
	// 錯誤步驟
	iErrorID	: INT;
	// 功能錯誤碼
	iFbErrorID	: INT;
	// 已歸零
	bHome	: BOOL;
	// 位置
	fPos : LREAL;
	
	b_ISVALIDREF : BOOL;
END_VAR

VAR_INPUT
	bJogMode: BOOL;
	// 移動軸
	Axis1: REFERENCE TO AXIS_REF;
	// 負極限
	inLimiter: BOOL;
	// 正極限
	outLimiter: BOOL;
	// 原點
	origin : BOOL;
	
	
END_VAR

IF __ISVALIDREF(Axis1) THEN
	b_ISVALIDREF := TRUE;
	Main();
END_IF

METHOD AbsMove : BOOL
VAR_INPUT
	// 目標位置
	_Position : LREAL;
	
	// 移動速度
	_Velocity : LREAL := 0;
END_VAR
bDone := FALSE;

Mode := ActionMode.AbsMove;
TargetPos := _Position;

IF _Velocity = 0 THEN
	Velocity := 10;
ELSE
	Velocity := _Velocity;
END_IF
// ============ 紀錄啟動條件 ============
_log.fbJson.StartObject();
_log.fbJson.AddKeyString('MethodName','AbsMove');
_log.fbJson.AddKeyLreal('Position', _Position);
_log.fbJson.AddKeyLreal('Velocity', _Velocity);
_log.JsonOutput();
// ======================================

step:=1;
END_METHOD

PROPERTY Axis_States : ST_AxisStatus
GET
Axis1.ReadStatus();
Axis_States := Axis1.Status;
END_GET
END_PROPERTY

METHOD Homing : BOOL
VAR
END_VAR
bDone := FALSE;
Mode := ActionMode.Home;

// ============ 紀錄啟動條件 ============
_log.fbJson.StartObject();
_log.fbJson.AddKeyString('MethodName','Homing');
_log.JsonOutput();
// ======================================


step:=1;
END_METHOD

ACTION Main:
Estop_Trig(CLK:= (SystemError OR Estop) AND Axis1.Status.Operational );

IF Estop_Trig.Q THEN
	iErrorId := step;
	step:=800;
	bDone := FALSE;
END_IF

bBuzy := step > 0 AND step < 10000;
berror := step >= 10000;
IF bBuzy OR berror THEN
	bDone := FALSE;
END_IF
IF bError THEN
	iErrorID := step - 10000;
	
END_IF

ws_step := INT_TO_WSTRING(step);

CASE step OF
	0://程式待命
		tmr1.IN					:= FALSE;
		tmr100.IN				:= FALSE;
		tmr200.IN				:= FALSE;
		tmr201.IN				:= FALSE;
		tmr800.IN				:= FALSE;
		tmrWdt.in 				:= FALSE;
		
END_CASE

IF step > 0 THEN
	Step0_Start();
	Step1_1_AbsMove();
	Step1_2_RelMove();
	Step1_3_Home();
	Step8_End();
END_IF

IF stepA > 0 THEN
	Step9_SetLimit();
END_IF

MC_FB();
fPos := LREAL_TO_REAL(Axis1.NcToPlc.ActPos);
timer();


move_RTrig(CLK := Axis1.Status.Moving);
move_FTrig(CLK := Axis1.Status.Moving);
IF move_RTrig.Q THEN
	move_Start_Pos := fPos;
END_IF 

IF move_FTrig.Q AND total_Move <> 0 THEN
	total_Move^ := total_Move^ + ABS(fPos - move_Start_Pos);
END_IF



_log(name:= TO_STRING(scAxisName), step:= step);
END_ACTION

ACTION MC_FB:
// 正轉極限
Axis1Power.Enable_Positive:= OutLimiter;
// 反轉極限
Axis1Power.Enable_Negative:= inLimiter;

Axis1.ReadStatus();

// 軸速度百分比
IF hmi.Auto_Pause THEN
	Axis1Power.Override := 0;
ELSE
	Axis1Power.Override := Axis.Override;
END_IF


(*===================== 軸電源 =====================*)
Axis1Power(Axis:= Axis1);


(*===================== 軸重置 =====================*)
Axis1Reset(Axis:= Axis1);


(*===================== 軸停止 =====================*)
Axis1Stop(Axis:= Axis1);


(*===================== 軸命令取消 =====================*)
Axis1Halt(Axis:= Axis1);


(*===================== 軸絕對移動 =====================*)
fb_AbsMove(Axis:= Axis1);


(*===================== 軸相對移動 =====================*)
fb_RelMove(Axis:= Axis1);

(*===================== 軸歸零 =====================*)
fb_Axis1_NcIoOutput(Axis:= Axis1, Device := NcIoDeviceDrive, NcIoOutput := NcIoOutputnCtrl2);

(*===================== 軸歸零 =====================*)
fb_Home(Axis:= Axis1, HomingMode:= MC_Direct);

(*===================== 軸寫入BOOL參數 =====================*)
fb_WriteBoolParameter(Axis:= Axis1);

(*===================== 軸寫入參數 =====================*)
fb_WriteParameter(Axis:= Axis1);

(*===================== 背隙補償 =====================*)
fb_BacklashCompensation(Axis:= Axis1);
END_ACTION

PROPERTY Name : WSTRING
GET
Name := scAxisName;
END_GET
SET
scAxisName := Name;
END_SET
END_PROPERTY

PROPERTY Pos : LREAL
GET
pos := fPos;
END_GET
END_PROPERTY

METHOD PowerOff : BOOL
VAR_INPUT
END_VAR
(*===============================
			關閉馬達
  ===============================*)

// ============ 紀錄啟動條件 ============
_log.fbJson.StartObject();
_log.fbJson.AddKeyString('MethodName','PowerOff');
_log.JsonOutput();
// ======================================


step:=800;
END_METHOD

METHOD PowerOn : BOOL
VAR_INPUT
END_VAR
bDone := FALSE;
Mode := ActionMode.DoNothing;



// ============ 紀錄啟動條件 ============
_log.fbJson.StartObject();
_log.fbJson.AddKeyString('MethodName','PowerOn');
_log.JsonOutput();
// ======================================


step:=1;
END_METHOD

METHOD RelMove : BOOL
VAR_INPUT
	// 目標位置
	_Position : LREAL;
	
	// 移動速度
	_Velocity : LREAL := 0;
END_VAR
bDone := FALSE;
Mode := ActionMode.RelMove;
TargetPos := _Position;

IF _Velocity = 0 THEN
	Velocity := 10;
ELSE
	Velocity := _Velocity;
END_IF


// ============ 紀錄啟動條件 ============
_log.fbJson.StartObject();
_log.fbJson.AddKeyString('MethodName','RelMove');
_log.fbJson.AddKeyLreal('Position', _Position);
_log.fbJson.AddKeyLreal('Velocity', _Velocity);
_log.JsonOutput();
// ======================================


step:=1;
END_METHOD

METHOD Set_Recoder : BOOL
VAR_INPUT
	total_Move_var : PVOID;
END_VAR
total_Move := total_Move_var;
END_METHOD

METHOD SetDyn : BOOL
VAR_INPUT
	SetJog : BOOL;
END_VAR
//IF SetJog THEN
// 	fb_AbsMove.Acceleration := 0;
// 	fb_AbsMove.Deceleration := 0;
// 	fb_RelMove.Acceleration := 0;
// 	fb_RelMove.Deceleration := 0;
//ELSE
//	fb_AbsMove.Acceleration := SpdC.DnZ_Accelerated;
//	fb_AbsMove.Deceleration := SpdC.DnZ_Deceleration;
//	fb_RelMove.Acceleration := SpdC.DnZ_Accelerated;
//	fb_RelMove.Deceleration := SpdC.DnZ_Deceleration;
//end_if
END_METHOD

METHOD SetLimit : BOOL
VAR_INPUT
END_VAR
stepA := 1;
END_METHOD

PROPERTY State : Sub_Step
GET
State.bBuzy := bBuzy;
State.bError := bError;
State.bDone := bDone;
State.Step := step;
END_GET
END_PROPERTY

ACTION Step0_Start:
	(*============================
				啟動馬達
	  ============================*)
CASE step OF
	
	1://開始移動流程
		// 設定狀態
		bDone := FALSE;
		tmrWdt.IN := FALSE;
//		SetDyn(bJogMode);
		Axis1Reset.Execute :=FALSE;
		_retry_count := 0;
		IF NOT bDone THEN
			step := 10;
		END_IF
		
	10:
		IF axis1.Status.Error THEN
			step := step + 1;
		ELSE
			step := 20;
		END_IF
		
	11:
		Axis1Reset.Execute :=TRUE;
		step := step + 1;
		
	12:
		IF NOT axis1.Status.Error AND Axis1Reset.Done THEN
			Axis1Reset.Execute :=FALSE;
			step := 20;
		ELSIF Axis1Reset.Error THEN
			pMsg.Push_Error(
					ErrorCodeConver.Str(str0:= scAxisName, str1:= ": 馬達無法重置", ErrorCode:= Axis1Reset.ErrorID)
			);
			Axis1Reset.Execute :=FALSE;
			step:=step + 10000;
		END_IF
		
	20: // 檢查馬達1是否已啟動
		IF NOT Axis1Power.Status  THEN
			step := step + 1;
		ELSE
			step := 60;
		END_IF
		
	21:// 啟動馬達1
		Axis1Power.Enable := TRUE;
		tmrWdt.IN := TRUE;
		step := step + 1;
		
	22:// 等待馬達啟動完成
		IF Axis1Power.Status THEN
			step := step + 1;
			tmrWdt.IN := FALSE;
			
		ELSIF tmrWdt.Q OR Axis1Power.Error THEN
			tmrWdt.IN := FALSE;
			IF _retry_count > 3 THEN
				pMsg.Push_Error(
						ErrorCodeConver.Str(str0:= scAxisName, str1:= ": 啟動失敗", ErrorCode:= Axis1Power.ErrorID)
				);
				step:=step + 10000;
			ELSE
				step := 10;
				_retry_count := _retry_count + 1;
			END_IF
		END_IF
		
	23:// 馬達啟動後延遲
		tmr1.in:=TRUE;
		IF tmr1.Q THEN
			tmr1.IN:=FALSE;
			step:=60;
		END_IF
		
	
			

	60: 
		fb_BacklashCompensation.Enable := FALSE;
		step := step + 1;
		
		
	61:	
		// 背隙值 (mm)
		fb_BacklashCompensation.Backlash := 0.05;
		// 正向補償 (往正方向移動時補償，預設是反方向移動時補償)
		fb_BacklashCompensation.CompensationInPositiveDirection := FALSE;
		// 背隙補償的速度 (mm/s)
		fb_BacklashCompensation.Ramp := 1;
		// 解除時機
		fb_BacklashCompensation.DisableMode  := E_DisableMode.DisableModeReset;
		// 功能啟動
		fb_BacklashCompensation.Enable := TRUE;
		step := step + 1;
		
	62:
		IF fb_BacklashCompensation.Enabled THEN
			step := step + 1;
		ELSIF fb_BacklashCompensation.Error THEN
			fb_BacklashCompensation.Enable := FALSE;
			step := step + 1;
		END_IF
		
	63:
		step := 80;
		
	80: //模式選擇
		CASE Mode OF
			ActionMode.AbsMove:
				step := 100;
				
			ActionMode.RelMove:
				step := 200;
				
			ActionMode.Home:
				step := 300;
				
			ActionMode.Find:
				step := 400;
				
			ActionMode.DoNothing:
				step := step + 1;
		END_CASE
		
	81:
		bdone := TRUE;
		step := 0;
		
END_CASE
END_ACTION

ACTION Step1_1_AbsMove:
	(*========================================
					開始移動
	=========================================*)	
CASE step OF
	100:
		fb_AbsMove.Execute := FALSE;
		Axis1Halt.Execute := FALSE;
		Axis1Stop.Execute := FALSE;
		step := step + 1;
		
	101:
		IF Velocity = 0 THEN
			pMsg.Push_Error( WStrConcat(str0:= scAxisName, str1:= ": Abs設定速度為0")
			);
		ELSE
			step := step + 1;
		END_IF
		
	102:
		IF fPos > TargetPos - 0.1 AND fPos < TargetPos + 0.1 THEN 
			step:= 190;
		ELSE
			step := step + 1;
		END_IF
		
	103:
		IF Axis1.Status.HasJob THEN
			Axis1Halt.Deceleration := 0;
			Axis1Halt.Execute := TRUE;
			step := step + 1;
		ELSE
			step:= 109;
		END_IF
		
	104:
		IF Axis1Halt.Busy OR Axis1Halt.Done OR Axis1Halt.Error THEN
			step:=step + 1;
		END_IF
		
	105:
		IF Axis1Halt.Done THEN
			Axis1Halt.Execute := FALSE;
			step:=step + 1;
		ELSIF Axis1Halt.Error THEN
			Axis1Halt.Execute := FALSE;
			step:=step + 10000;
		END_IF
		
	106:
		step:= 109;
		
	109:
		step:= 110;
		

	110: // 設定移動位置
		fb_AbsMove.Position := TargetPos;
		fb_AbsMove.Velocity:= Velocity;
		fb_AbsMove.BufferMode:= MC_Aborting;
		step:=step + 1;
		
	111:
		fb_AbsMove.Execute := TRUE;
		step:=step + 1;
		
	112:
		IF fb_AbsMove.Busy OR fb_AbsMove.Done OR fb_AbsMove.Error THEN
			step:=step + 1;
		END_IF
		
	113:
		IF fb_AbsMove.Done OR (TargetPos <= 0 AND pos < 2 AND Origin) THEN
			fb_AbsMove.Execute := FALSE;
			step:=step + 1;
		ELSIF fb_AbsMove.Error THEN
			pMsg.Push_Error(
				ErrorCodeConver.Str(str0:= scAxisName, str1:= ": Abs移動失敗", ErrorCode:= fb_AbsMove.ErrorID)
			);
			fb_AbsMove.Execute := FALSE;
			step:=step + 10000;
		END_IF
		
	114:
		step := 190;
		
	190:
		bDone := TRUE;
		step:=890;
END_CASE
END_ACTION

ACTION Step1_2_RelMove:
	(*========================================
					開始移動
	=========================================*)	
CASE step OF
	200:
		fb_RelMove.Execute := FALSE;
		Axis1Halt.Execute := FALSE;
		Axis1Stop.Execute := FALSE;
		step := step + 1;
		
	201:
		IF Velocity = 0 THEN
			pMsg.Push_Error(
				WStrConcat(scAxisName, ":Rel設定速度為0")
			);
		ELSE
			step := step + 1;
		END_IF
		
	202:
		IF TargetPos = 0 THEN 
			step:= 280;
		ELSE
			step := step + 1;
		END_IF
		
	203:
		IF Axis1.Status.HasJob THEN
			Axis1Halt.Deceleration := 0;
			Axis1Halt.Execute := TRUE;
			step := step + 1;
		ELSE
			step:= 209;
		END_IF
		
	204:
		IF Axis1Halt.Busy OR Axis1Halt.Done OR Axis1Halt.Error THEN
			step:=step + 1;
		END_IF
		
	205:
		IF Axis1Halt.Done THEN
			Axis1Halt.Execute := FALSE;
			step:=step + 1;
		ELSIF Axis1Halt.Error THEN
			Axis1Halt.Execute := FALSE;
			step:=step + 10000;
		END_IF
		
	206:
		step:= 209;
		
	209:
		step:= 210;
		

	210: // 設定移動位置
		fb_RelMove.Distance := TargetPos;
		fb_RelMove.Velocity:= Velocity;
		fb_RelMove.BufferMode:= MC_Aborting;
		step:=step + 1;
		
	211:
		fb_RelMove.Execute := TRUE;
		step:=step + 1;
		
	212:
		IF fb_RelMove.Busy OR fb_RelMove.Done OR fb_RelMove.Error THEN
			step:=step + 1;
		END_IF
		
	213:
		IF fb_RelMove.Done THEN
			fb_RelMove.Execute := FALSE;
			step:=step + 1;
		ELSIF fb_RelMove.Error THEN
			pMsg.Push_Error(
				ErrorCodeConver.Str(str0:= scAxisName, str1:= ":Rel移動失敗", ErrorCode:= fb_RelMove.ErrorID)
			);
			fb_RelMove.Execute := FALSE;
			step:=step + 10000;
		END_IF
		
	214:
		step:=290;
		
	280:
		tmr1.PT := T#500MS;
		tmr1.IN := TRUE;
		IF tmr1.Q THEN
			tmr1.IN := FALSE;
			step:=step + 1;
		END_IF
		
	281:
		step := 290;
		
	290:
		bDone := TRUE;
		step:=890;
END_CASE
END_ACTION

ACTION Step1_3_Home:
(*========================================
				歸零
=========================================*)	
CASE step OF
	300:
		fb_Axis1_NcIoOutput.Execute := FALSE;
		fb_Home.Execute := FALSE;
		step := step + 1;
		
	301: // 關閉負軟體極限
		fb_WriteBoolParameter.ParameterNumber := MC_AxisParameter.EnableLimitNeg;
		fb_WriteBoolParameter.Value := FALSE;
		fb_WriteBoolParameter.Execute := TRUE;
		step := step + 1;
		
	302:
		IF fb_WriteBoolParameter.Done OR fb_WriteBoolParameter.Error THEN
			fb_WriteBoolParameter.Execute := FALSE;
			IF fb_WriteBoolParameter.Error THEN
				pMsg.Push_Alarm_NoPause(
					ErrorCodeConver.Str(str0:= scAxisName, str1:= ": 寫入 使用負方向極限 參數發生錯誤", str2:= ws_step, ErrorCode := fb_WriteBoolParameter.ErrorID)
					);
			END_IF
			step := step + 1;
		END_IF
	
	303:
		Origin_pos := Pos;
		step:= 340;
		
// 	310: // 尋找負極限訊號
// 		fb_RelMove.Distance := -9999;
// 		fb_RelMove.Velocity:= 1;
// 		fb_RelMove.BufferMode:= MC_Aborting;
// 		fb_RelMove.Execute := TRUE;
// 		step:=step + 1;
// 		
// 	311:
// 		IF fb_RelMove.Busy OR fb_RelMove.Error THEN
// 			fb_RelMove.Execute := FALSE;
// 			step:=step + 1;
// 		END_IF
// 		
// 	312:
// 		IF NOT inLimiter THEN
// 			Axis1Halt.Execute := TRUE;
// 			step:=step + 1;
// 		ELSIF fb_RelMove.Done THEN
// 			pmsg.Push_Error(ErrorCodeConver.Str2(scAxisName, ":無法找到負極限訊號", 0));
// 			step:=step + 10000;
// 		ELSIF fb_RelMove.Error THEN
// 			pmsg.Push_Error(ErrorCodeConver.Str2(scAxisName, ":歸零移動時發生錯誤", fb_RelMove.ErrorID));
// 			step:=step + 10000;
// 		END_IF
// 		
// 	313:
// 		IF Axis1Halt.Busy OR Axis1Halt.Error THEN
// 			Axis1Halt.Execute := FALSE;
// 			step:=step + 1;
// 		END_IF
// 		
// 	314:
// 		IF Axis1Halt.Done THEN
// 			step:=step + 1;
// 		ELSIF Axis1Halt.Error THEN
// 			pmsg.Push_Error(ErrorCodeConver.Str2(scAxisName, ":取消軸移動命令時發生錯誤", Axis1Halt.ErrorID));
// 			step:=step + 10000;
// 		END_IF
// 		
// 	315:
// 		tmr200.in :=TRUE;
// 		IF tmr200.q THEN
// 			tmr200.in :=FALSE;
// 			step := step + 1;
// 		END_IF
// 		
// 	316:
// 		step := 320;
// 		
// 		
// 	320: // 脫離負極限
// 		fb_RelMove.Distance := 9999;
// 		fb_RelMove.Velocity:= 0.005;
// 		fb_RelMove.BufferMode:= MC_Aborting;
// 		fb_RelMove.Execute := TRUE;
// 		step:=step + 1;
// 		
// 	321:
// 		IF fb_RelMove.Busy OR fb_RelMove.Error THEN
// 			fb_RelMove.Execute := FALSE;
// 			step:=step + 1;
// 		END_IF
// 		
// 	322:
// 		IF inLimiter THEN
// 			Axis1Halt.Execute := TRUE;
// 			step:=step + 1;
// 		ELSIF fb_RelMove.Done THEN
// 			pmsg.Push_Error(ErrorCodeConver.Str2(scAxisName, ":無法找到負極限訊號", 0));
// 			step:=step + 10000;
// 		ELSIF fb_RelMove.Error THEN
// 			pmsg.Push_Error(ErrorCodeConver.Str2(scAxisName, ":歸零移動時發生錯誤", fb_RelMove.ErrorID));
// 			step:=step + 10000;
// 		END_IF
// 		
// 	323:
// 		IF Axis1Halt.Busy OR Axis1Halt.Error THEN
// 			Axis1Halt.Execute := FALSE;
// 			step:=step + 1;
// 		END_IF
// 		
// 	324:
// 		IF Axis1Halt.Done THEN
// 			step:=step + 1;
// 		ELSIF Axis1Halt.Error THEN
// 			pmsg.Push_Error(ErrorCodeConver.Str2(scAxisName, ":取消軸移動命令時發生錯誤", Axis1Halt.ErrorID));
// 			step:=step + 10000;
// 		END_IF
// 		
// 	325:
// 		tmr200.in :=TRUE;
// 		IF tmr200.q THEN
// 			tmr200.in :=FALSE;
// 			step := step + 1;
// 		END_IF
// 		
// 	326:
// 		step := 330;
// 		
// 	330:
// 		fb_RelMove.Distance := 2;
// 		fb_RelMove.Velocity:= 2;
// 		fb_RelMove.BufferMode:= MC_Aborting;
// 		fb_RelMove.Execute := TRUE;
// 		step:=step + 1;
// 		
// 	331:
// 		IF fb_RelMove.Busy OR fb_RelMove.Error THEN
// 			fb_RelMove.Execute := FALSE;
// 			step:=step + 1;
// 		END_IF
// 		
// 	332:
// 		IF fb_RelMove.Done THEN
// 			step:=step + 1;
// 		ELSIF fb_RelMove.Error THEN
// 			pmsg.Push_Error(ErrorCodeConver.Str2(scAxisName, ":歸零移動時發生錯誤", fb_RelMove.ErrorID));
// 			step:=step + 10000;
// 		END_IF
// 		
// 	333:
// 		tmr200.in :=TRUE;
// 		IF tmr200.q THEN
// 			tmr200.in :=FALSE;
// 			step := step + 1;
// 		END_IF
// 		
// 	334:
// 		step := 350;
		
	340:
		fb_Axis1_NcIoOutput.BitSelectMask := 128;
		fb_Axis1_NcIoOutput.BitValues := 128;
		fb_Axis1_NcIoOutput.Execute := TRUE;
		IF fb_Axis1_NcIoOutput.Done THEN
			step := step + 1;
			fb_Axis1_NcIoOutput.Execute := FALSE;
		ELSIF fb_Axis1_NcIoOutput.Error THEN
			pMsg.Push_Error(
				ErrorCodeConver.Str(str0:= scAxisName, str1:= ":Home寫入驅動器失敗", str2:= ws_step, ErrorCode := fb_Axis1_NcIoOutput.ErrorID)
			);
			fb_Axis1_NcIoOutput.Execute := FALSE;
			step:=step + 10000;
		END_IF
		
	341:
		fb_Axis1_NcIoOutput.BitSelectMask := 128;
		fb_Axis1_NcIoOutput.BitValues := 0;
		fb_Axis1_NcIoOutput.Execute := TRUE;
		IF fb_Axis1_NcIoOutput.Done THEN
			step := step + 1;
			fb_Axis1_NcIoOutput.Execute := FALSE;
		ELSIF fb_Axis1_NcIoOutput.Error THEN
			pMsg.Push_Error(
				ErrorCodeConver.Str(str0:= scAxisName, str1:= ":Home寫入驅動器失敗", str2:= ws_step, ErrorCode := fb_Axis1_NcIoOutput.ErrorID)
			);
			fb_Axis1_NcIoOutput.Execute := FALSE;
			step:=step + 10000;
		END_IF
		
	342:
		tmr200.in :=TRUE;
		IF tmr200.q THEN
			tmr200.in :=FALSE;
			step := step + 1;
		END_IF
		
	343:
		Axis1Power.Enable := FALSE;
		tmrWdt.IN := TRUE;
		IF NOT Axis1Power.Status THEN
			step := step + 1;
			tmrWdt.IN := FALSE;
			
		ELSIF tmrWdt.Q OR Axis1Power.Error THEN
			pMsg.Push_Error(
				ErrorCodeConver.Str(str0:= scAxisName, str1:= ":關閉失敗", str2:= ws_step, ErrorCode := Axis1Power.ErrorID)
			);
			step:=step + 10000;
		END_IF	
		
	344:
		tmr200.in :=TRUE;
		IF tmr200.q THEN
			tmr200.in :=FALSE;
			step := step + 1;
		END_IF
		
	345:
		step:= 350;
		
	
			
		
	350:// 設定原點
		fb_Home.Execute := TRUE;
		step:=step + 1;
		
	351:
		IF fb_Home.Done THEN
			fb_Home.Execute := FALSE;
			bHome := TRUE;
			step:=step + 1;
		ELSIF fb_Home.Error THEN
			pMsg.Push_Error(
				ErrorCodeConver.Str(str0:= scAxisName, str1:= ":位置清除失敗", str2:= ws_step, ErrorCode := fb_Home.ErrorID)
			);
			fb_Home.Execute := FALSE;
			step:=step + 10000;
		END_IF
		
	352:
		Axis1Power.Enable := TRUE;
		tmrWdt.IN := TRUE;
		IF Axis1Power.Status THEN
			step := step + 1;
			tmrWdt.IN := FALSE;
		ELSIF tmrWdt.Q OR Axis1Power.Error THEN
			pMsg.Push_Error(
				ErrorCodeConver.Str(str0:= scAxisName, str1:= ":啟動失敗", str2:= ws_step, ErrorCode := Axis1Power.ErrorID)
			);
			step:=step + 10000;
		END_IF	
			
	353:
		tmr200.in :=TRUE;
		IF tmr200.q THEN
			tmr200.in :=FALSE;
			step:=step + 1;
		END_IF
		
	354:
		step:= 360;
		
	360:// 設定移動位置
		step:= 390;
	
			
	390://延遲
		tmr200.in :=TRUE;
		IF tmr200.q THEN
			tmr200.in :=FALSE;
			bDone := TRUE;
			step:=890;
		END_IF
END_CASE
END_ACTION

ACTION Step8_End:
	(*======================================
					關閉馬達
	  ======================================*)
CASE step OF
	800:
		Axis1Reset.Execute	:= FALSE;
		Axis1Stop.Execute	:= FALSE;
		Axis1Halt.Execute	:= FALSE;
		fb_AbsMove.Execute	:=FALSE;
		fb_RelMove.Execute	:=FALSE;
		fb_Home.Execute		:=FALSE;
		step := step + 1;
			
	// ============== 停止 + 關閉==============
	801:
		IF Axis1.Status.Moving THEN
			step := step + 1;
		ELSE
			step := 810;
		END_IF
	
	802:
		Axis1Stop.Execute := TRUE;
		step := step + 1;
		
	803:
		Axis1Stop.Execute := TRUE;
		step := step + 1;
		
	804:
		IF Axis1Stop.Done OR Axis1Stop.Error THEN
			Axis1Stop.Execute := FALSE;
			step := step + 1;
		END_IF
		
	805:
		tmr800.PT := T#1S;
		tmr800.in:=TRUE;
		IF tmr800.Q THEN
			tmr800.IN:=FALSE;
			step := step + 1;
		END_IF
		
	806:
		step:=810;
		
	810:
		Axis1Power.Enable := FALSE;
		IF Axis1.Status.Disabled THEN
			step := step + 1;
		END_IF
		
			
	811:// 馬達關閉後延遲
		tmr800.in:=TRUE;
		IF tmr800.Q THEN
			tmr800.IN:=FALSE;
			step := step + 1;
		END_IF
		
	812:
		Mode := ActionMode.DoNothing;
		step:=890;
		
		
// ==============停止==============
	850:
		Axis1Stop.Deceleration := Dec;
		Axis1Stop.Execute := FALSE;
		step := step + 1;
		
	851:
		Axis1Stop.Execute := TRUE;
		step := step + 1;
		
	852:
		IF Axis1Stop.Done OR Axis1Stop.Error THEN
			Axis1Stop.Execute := FALSE;
			step := step + 1;
		END_IF
		
	853:
		tmr800.PT := T#1S;
		tmr800.in:=TRUE;
		IF tmr800.Q THEN
			tmr800.IN:=FALSE;
			step := step + 1;
		END_IF
		
	854:
		step:=890;
		
		
			
	890:// 結束程式
		Mode := ActionMode.DoNothing;
		step:=0;

END_CASE
END_ACTION

ACTION Step9_SetLimit:
CASE stepA OF
	1:
		fb_WriteParameter.Execute := FALSE;
		fb_WriteBoolParameter.Execute := FALSE;
		stepA := stepA + 1;
		
	2:
		stepA := 10;
	
(* ================ 設定正方向極限 ================ *)		
		
	10: // 設定是否使用 正方向極限 數值為0設為false
		fb_WriteBoolParameter.ParameterNumber := MC_AxisParameter.EnableLimitPos;
		fb_WriteBoolParameter.Value := PosC.GaX_P_Limite <> 0;
		fb_WriteBoolParameter.Execute := TRUE;
		stepA := stepA + 1;
		
		
	11:
		IF fb_WriteBoolParameter.Done OR fb_WriteBoolParameter.Error THEN
			fb_WriteBoolParameter.Execute := FALSE;
			IF fb_WriteBoolParameter.Error THEN
				pMsg.Push_Alarm_NoPause(
					ErrorCodeConver.Str(str0:= scAxisName, str1:= ": 寫入 使用正方向極限 參數發生錯誤", ErrorCode:= fb_WriteBoolParameter.ErrorID)
					);
			END_IF
			stepA := stepA + 1;
		END_IF
		
	12:
		IF PosC.GaX_P_Limite <> 0 THEN
			stepA := 20;
		ELSE
			stepA := 30;
		END_IF
			
		
	20: // 設定正方向極限
		fb_WriteParameter.ParameterNumber := MC_AxisParameter.SWLimitPos;
		fb_WriteParameter.Value := REAL_TO_LREAL(PosC.GaX_P_Limite);
		fb_WriteParameter.Execute := TRUE;
		stepA := stepA + 1;
		
		
	21:
		IF fb_WriteParameter.Done OR fb_WriteParameter.Error THEN
			fb_WriteParameter.Execute := FALSE;
			IF fb_WriteParameter.Error THEN
				pMsg.Push_Alarm_NoPause(
					ErrorCodeConver.Str(str0:= scAxisName, str1:= ": 寫入 正方向極限位置 參數發生錯誤", ErrorCode:= fb_WriteParameter.ErrorID)
					);
			END_IF
			stepA := stepA + 1;
		END_IF
		
	22:
		stepA := 30;
		
(* ================ 設定負方向極限 ================ *)		
		
	30: // 設定是否使用 負方向極限 數值為0設為false
		fb_WriteBoolParameter.ParameterNumber := MC_AxisParameter.EnableLimitNeg;
		fb_WriteBoolParameter.Value := PosC.GaX_N_Limite <> 0;
		fb_WriteBoolParameter.Execute := TRUE;
		stepA := stepA + 1;
		
		
	31:
		IF fb_WriteBoolParameter.Done OR fb_WriteBoolParameter.Error THEN
			fb_WriteBoolParameter.Execute := FALSE;
			IF fb_WriteBoolParameter.Error THEN
				pMsg.Push_Alarm_NoPause(
					ErrorCodeConver.Str(str0:= scAxisName, str1:= ": 寫入 使用負方向極限 參數發生錯誤", ErrorCode:= fb_WriteBoolParameter.ErrorID)
					);
			END_IF
			stepA := stepA + 1;
		END_IF
		
	32:
		IF PosC.GaX_N_Limite <> 0 THEN
			stepA := 40;
		ELSE
			stepA := 50;
		END_IF
			
		
	40: // 設定負方向極限
		fb_WriteParameter.ParameterNumber := MC_AxisParameter.SWLimitNeg;
		fb_WriteParameter.Value := REAL_TO_LREAL(PosC.GaX_N_Limite);
		fb_WriteParameter.Execute := TRUE;
		stepA := stepA + 1;
		
		
	41:
		IF fb_WriteParameter.Done OR fb_WriteParameter.Error THEN
			fb_WriteParameter.Execute := FALSE;
			IF fb_WriteParameter.Error THEN
				pMsg.Push_Alarm_NoPause(
					ErrorCodeConver.Str(str0:= scAxisName, str1:= ": 寫入 負方向極限位置 參數發生錯誤", ErrorCode:= fb_WriteParameter.ErrorID)
					);
			END_IF
			stepA := stepA + 1;
		END_IF
		
	42:
		stepA := 50;
		
(* ================ 設定結束 ================ *)	
	50:
		stepA := 0;
		
END_CASE
END_ACTION

METHOD Stop : BOOL
VAR_INPUT
	Dec : LREAL := 0;
END_VAR
(*===============================
			關閉馬達
  ===============================*)


// ============ 紀錄啟動條件 ============
_log.fbJson.StartObject();
_log.fbJson.AddKeyString('MethodName','Stop');
_log.fbJson.AddKeyLreal('Dec', Dec);
_log.JsonOutput();
// ======================================


step:=850;
END_METHOD

ACTION timer:
tmr1();
tmr2();
tmr100(PT:=T#50MS);
tmr200();
tmr201();
tmr800();
tmrWdt();
END_ACTION

END_FUNCTION_BLOCK

// ---- MSG/通知訊息/uuidv7_g.TcPOU
PROGRAM uuidv7_g
VAR
	fbStartProcess : NT_StartProcess;
	step: INT;
END_VAR
VAR_OUTPUT
	bBuzy : BOOL;
	bDone : BOOL;
	bError : BOOL;
	UUID:STRING(36);
	ErrorID : UDINT;
END_VAR

CASE step OF
	1:
		UUID := '';
		fbStartProcess.START := FALSE;
		step := step + 1;
		
	2:
		fbStartProcess.START := TRUE;
		step := step + 1;
		
	3:
		IF fbStartProcess.BUSY OR fbStartProcess.ERR THEN
			step := step + 1;
		END_IF
		
	4:
		IF NOT fbStartProcess.BUSY AND NOT fbStartProcess.ERR THEN
			fbStartProcess.START := FALSE;
			step := step + 1;
		ELSIF fbStartProcess.ERR THEN
			fbStartProcess.START := FALSE;
			ErrorID := fbStartProcess.ERRID;
			step := step + 10000;
		END_IF
		
	5:
		IF Len(UUID) >= 36 THEN
			bDone := TRUE;
			step := 0;
		END_IF
END_CASE
	

bBuzy := step > 0 AND step < 10000;

bError := step > 10000;

IF bBuzy THEN
	bDone := FALSE;
END_IF

fbStartProcess(
		NETID := '',
		PATHSTR := 'C:\custom\uuidv7generator_ads\uuidv7generator_ads.exe',
		DIRNAME := 'C:\custom\uuidv7generator_ads',
		COMNDLINE := '127.0.0.1.1.1 851 uuidv7_g.UUID',
		TMOUT := T#1S
	);

METHOD Get
VAR_INPUT
END_VAR
step := 1;
END_METHOD

END_PROGRAM

// ---- POUs/功能塊/RW_Config.TcPOU
PROGRAM RW_Config
VAR
	File_Path: STRING(INT#80) := '\Hard Disk2\Config\';
	fb_recipemancommands:recipemancommands;
	result: ARRAY [0..6] OF DWORD;
	result1: BOOL;
	boot: BOOL := true;
	



	GetTime: FB_LocalSystemTime := (bEnable := TRUE);
	

	tmr2: TON;
	tmr3: TON;
	
	//	目前時間	
	TimeNow: DATE_AND_TIME;
	
	strTimeNow: STRING;
END_VAR

VAR_INPUT
	// 寫入檔案
	Wrtie: BOOL;
END_VAR

tmr2(in:=boot, PT:=T#5S);
tmr3(in:=result1, PT:=T#1S);
IF tmr2.Q THEN
	result1 := fb_recipemancommands.SetStoragePath(File_Path);
	IF  tmr3.Q THEN
//		result[0] := fb_recipemancommands.LoadAndWriteRecipe('Config','Diff');
//		IF result[0] <> 0 THEN
//			result[1] := fb_recipemancommands.LoadRecipe('Config','Diff');
//			result[2] := fb_recipemancommands.WriteRecipe('Config','Diff');
//		END_IF
//		result1 := FALSE;
		boot := FALSE;
		Wrtie := TRUE;
	END_IF
END_IF

IF Wrtie THEN
	result1 := fb_recipemancommands.SetStoragePath(File_Path);
	result[3] := fb_recipemancommands.ReadRecipe('Config', 'Diff');
	result[4] := fb_recipemancommands.SaveRecipe('Config', 'Diff');
	result[5] := fb_recipemancommands.ReadAndSaveAs('Config','Diff');
	result[6] := fb_recipemancommands.ReadAndSaveRecipeAs('Config', 'Diff', CONCAT(STR1:= 'config_', STR2:= strTimeNow));
	Wrtie := FALSE;
END_IF



GetTime();
TimeNow:=SYSTEMTIME_TO_DT(GetTime.systemTime);
strTimeNow := CONCAT(STR1:= WORD_TO_STRING(GetTime.systemTime.wYear), STR2:='_');
strTimeNow := CONCAT(strTimeNow ,CONCAT(STR1:= WORD_TO_STRING(GetTime.systemTime.wMonth), STR2:='_'));
strTimeNow := CONCAT(strTimeNow ,CONCAT(STR1:= WORD_TO_STRING(GetTime.systemTime.wDay), STR2:='_'));
strTimeNow := CONCAT(strTimeNow ,WORD_TO_STRING(GetTime.systemTime.wHour));

END_PROGRAM

// ---- POUs/功能塊/字串處理功能塊/字串填充/FILLSTRING.TcPOU
FUNCTION FILLSTRING : STRING
VAR_INPUT
	str : STRING;
	strlen : INT;
	fill_char : STRING(1);
END_VAR
VAR
	rawlen : INT;
	
	fillNumber : INT;
	
	tmpstr : STRING;
	
	i : INT;
END_VAR

rawlen := LEN(STR:= str);

fillNumber := strlen - rawlen;

tmpstr := '';

FOR i:= 1 TO fillNumber DO
	tmpstr := CONCAT(STR1:= tmpstr, STR2:= fill_char);
END_FOR

FILLSTRING := CONCAT(STR1:= tmpstr, STR2:= str);

END_FUNCTION

// ---- POUs/功能塊/字串處理功能塊/浮點轉字串控制去小數點/Real2String.TcPOU
FUNCTION Real2String : STRING
VAR_INPUT
	num : LREAL;
	strlen : INT := 2;
END_VAR
VAR
	_pointPos : INT;
	
	fillNumber : INT;
	
	tmpstr : STRING;
	
	i : INT;
END_VAR

tmpstr := TO_STRING(num);

_pointPos := FIND(tmpstr, '.') + strlen;

Real2String := LEFT(tmpstr, _pointPos);

END_FUNCTION

// ---- POUs/功能塊/字串處理功能塊/字串連接/StrConcat.TcPOU
FUNCTION StrConcat : STRING(511)
VAR_INPUT
	str0 : STRING(511) := '';
	str1 : STRING(511) := '';
	str2 : STRING(511) := '';
	str3 : STRING(511) := '';
	str4 : STRING(511) := '';
	str5 : STRING(511) := '';
	str6 : STRING(511) := '';
	str7 : STRING(511) := '';
	str8 : STRING(511) := '';
END_VAR
VAR
	tmpstr : STRING(511);
END_VAR

tmpstr := CONCAT(STR1:= str0, STR2:= str1);
tmpstr := CONCAT(STR1:= tmpstr, STR2:= str2);
tmpstr := CONCAT(STR1:= tmpstr, STR2:= str3);
tmpstr := CONCAT(STR1:= tmpstr, STR2:= str4);
tmpstr := CONCAT(STR1:= tmpstr, STR2:= str5);
tmpstr := CONCAT(STR1:= tmpstr, STR2:= str6);
tmpstr := CONCAT(STR1:= tmpstr, STR2:= str7);
tmpstr := CONCAT(STR1:= tmpstr, STR2:= str8);
StrConcat := tmpstr;
RETURN;

END_FUNCTION

// ---- POUs/功能塊/資料庫 Postgre相關/記錄用/程式紀錄/Step_Log_Clear.TcPOU
PROGRAM Step_Log_Clear
VAR
	db_fb_PLCDBCmdEvt : FB_PLCDBCmdEvt(sNetID:= '', tTimeout:= T#5S );
	
	_stPara		: ARRAY [0..3] OF ST_ExpParameter;
	
	_SqlCommand : STRING(1024);
	
	_extrasstr : STRING(255);
	
	_fbJson      : FB_JsonSaxWriter;
	Clear_date: LINT;
END_VAR

Clear_date := TO_LINT(F_GetSystemTime());

// SQL命令
_SqlCommand := 

'DELETE 
	INTO program_running_log 
		(program_name, step_number, created_at, detail_data)
	VALUES
		({program_name}, {step_number}, to_timestamp(({created_at} - 116444736000000000) / 10000000.0), {detail_data}::jsonb);
';


db_fb_PLCDBCmdEvt.Execute(
	hDBID := 3,
	pExpression := ADR(_SqlCommand),			// SQL 命令 ex. SELECT * FROM PlcTest.newtable WHERE ID = {ID}  
	cbExpression := SIZEOF(_SqlCommand),		// SQL 命令字串的長度
	pData:= 0,		// 帶入的參數值
	cbData:= 0,//itmp, 	// 帶入的參數值大小
	pParameter:= 0, 				// 帶入的參數類型設定  ex.上面命令內的 {ID} 類型設定
	cbParameter:= 0,			// 帶入的參數類型設定的大小
)

{attribute 'suppress_wrn_C0410'}
PROPERTY fbJson : REFERENCE TO FB_JsonSaxWriter
GET
fbJson REF= _fbJson;
END_GET
END_PROPERTY

METHOD JsonOutput : BOOL
VAR_INPUT
END_VAR
fbJson.EndObject();
_extrasstr := fbJson.GetDocument();
fbJson.ResetDocument();
END_METHOD

END_PROGRAM

// ---- POUs/硬體控制/其他控制/螢幕旋轉/TurnMonitor.TcPOU
PROGRAM TurnMonitor
VAR
	MonitorSensor_RTrig : R_trig;
	MonitorSensor_FTrig : F_trig;
	
	winCmd: NT_StartProcess := (NETID := '192.168.31.180.1.1');
	
	turn270: BOOL;
	turn0: BOOL;
END_VAR

MonitorSensor_RTrig(CLK := IO.i207);
MonitorSensor_FTrig(CLK := IO.i207);

IF MonitorSensor_RTrig OR turn270 THEN 
	turn270 := FALSE;
	winCmd.DIRNAME := 'C:\Users\MyUser\Documents\multimonitortool-x64';
	winCmd.PATHSTR := 'C:\Users\MyUser\Documents\multimonitortool-x64\MultiMonitorTool.exe';
	winCmd.COMNDLINE := '/SetOrientation 1 270';
	winCmd.START := TRUE;
END_IF

IF MonitorSensor_RTrig OR turn0 THEN 
	turn270 := FALSE;
	winCmd.DIRNAME := 'C:\Users\MyUser\Documents\multimonitortool-x64';
	winCmd.PATHSTR := 'C:\Users\MyUser\Documents\multimonitortool-x64\MultiMonitorTool.exe';
	winCmd.COMNDLINE := '/SetOrientation 1 0';
	winCmd.START := TRUE;
END_IF


IF NOT winCmd.BUSY THEN
	winCmd := FALSE;
END_IF

END_PROGRAM

// ---- POUs/硬體控制/測距感應器/DT80_Decoder.TcPOU
FUNCTION_BLOCK DT80_Decoder IMPLEMENTS I_DisSensor
VAR_INPUT
	// 關閉感應器
	DisableSeosor :	BOOL;
END_VAR
VAR_OUTPUT
	// 距離 (單位:mm)
	fDistance : LREAL;
	// 裝置狀態正常
	SSC1_1			:BOOL;
	// 裝置狀態正常
	bDevice_is_OK			:BOOL;
	// 需要維護
	bMaintenance_required	:BOOL;
	// 超出測量距離
	bOut_of_specification	:BOOL;
	// 檢查功能
	bFunctional_check		:BOOL;
	// 錯誤
	bFailure				:BOOL;
	// 距離比例(單位:公尺)
	iScale_Distance			:INT;
END_VAR
VAR
	// 原始資料輸入
	in_RawData AT %I* : ARRAY [0..7] OF USINT;
	// 原始資料輸出
	out_rawdata AT %Q* :USINT;	
	
	

	DistanceTmp : DINT;
	
	tmpfDistance : POINTER TO SINT;
END_VAR

fDistance := (in_RawData[0] * EXPT(2, 24)) + (in_RawData[1] * EXPT(2, 16)) + (in_RawData[2] * EXPT(2, 8)) + (in_RawData[3] * EXPT(2, 0));
tmpfDistance := ADR(in_RawData[4]);

fDistance := fDistance * EXPT(10, tmpfDistance^);

PROPERTY Distance : LREAL
GET
Distance := fDistance;
END_GET
END_PROPERTY

END_FUNCTION_BLOCK
